FUNCTION_BLOCK print
  (* Standard: 61499-2 *)
  (* Version 0.1, 2018-00-07, hpea485, UOA *)
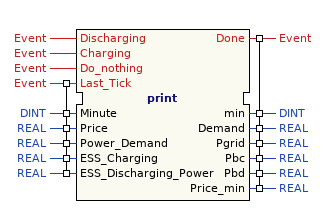
  EVENT_INPUT
    Discharging;
    Charging;
    Do_nothing;
    Last_Tick WITH Minute, Price, Power_Demand, ESS_Charging, ESS_Discharging_Power;
  END_EVENT
  EVENT_OUTPUT
    Done WITH min, Demand, Pgrid, Pbc, Pbd, Price_min;
  END_EVENT
  VAR_INPUT
    Minute : DINT;
    Price : REAL;
    Power_Demand : REAL;
    ESS_Charging : REAL;
    ESS_Discharging_Power : REAL;
  END_VAR
  VAR_OUTPUT
    min : DINT;
    Demand : REAL;
    Pgrid : REAL;
    Pbc : REAL;
    Pbd : REAL;
    Price_min : REAL;
  END_VAR
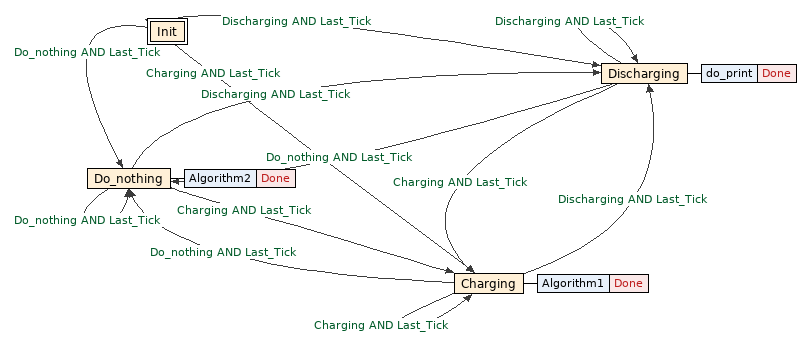
  EC_STATES
    Init;
    Do_nothing : Algorithm2 -> Done;
    Discharging : do_print -> Done;
    Charging : Algorithm1 -> Done;
  END_STATES
  EC_TRANSITIONS
    Do_nothing TO Discharging := Discharging AND Last_Tick;
    Do_nothing TO Charging := Charging AND Last_Tick;
    Do_nothing TO Do_nothing := Do_nothing AND Last_Tick;
    Discharging TO Charging := Charging AND Last_Tick;
    Discharging TO Do_nothing := Do_nothing AND Last_Tick;
    Discharging TO Discharging := Discharging AND Last_Tick;
    Charging TO Discharging := Discharging AND Last_Tick;
    Charging TO Do_nothing := Do_nothing AND Last_Tick;
    Charging TO Charging := Charging AND Last_Tick;
    Init TO Do_nothing := Do_nothing AND Last_Tick;
    Init TO Discharging := Discharging AND Last_Tick;
    Init TO Charging := Charging AND Last_Tick;
  END_TRANSITIONS
  ALGORITHM do_print IN C:
REAL ESS = me->ESS_Discharging_Power;
REAL Pg = me->Power_Demand - ESS;
REAL Power_Demand = me->Power_Demand;
REAL the_price = me->Price;
DINT minute = me->Minute;
printf("Minute in soc do_print %d \r\n", minute);
printf("the price do_print %f \r\n", the_price);
//if (Power_Demand == ESS){
//the_price = 0;
//}
//else if(Power_Demand == Pg){
//the_price = Pg * me->Price;
//}
me->min = minute;
me->Demand = Power_Demand;
me->Pgrid= Pg;
me->Pbc = 0;
me->Pbd = ESS;
me->Price_min = the_price / (30* 2* 1000);// converting $/Mwh to $/kwmin

printf("--------OUTPUT DISCHARGING STATE ------  \r\n");
//printf("DONE \r\n");
printf("Current Minute: %d\tCurrent Price:%f\r\n", me->Minute, the_price);
  END_ALGORITHM
  ALGORITHM Algorithm1 IN C:
REAL the_price = me->Price;
REAL ESS = 200;
REAL Pg = me->Power_Demand + ESS;
REAL Power_Demand = me->Power_Demand;
DINT minute = me->Minute;

me->min = minute;
me->Demand = Power_Demand;
me->Pgrid= Pg;
me->Pbc = ESS;
me->Pbd = 0;
me->Price_min = the_price / (30* 2* 1000);// converting $/Mwh to $/kwmin
printf("Minute in soc al1 %d \r\n", minute);


printf("-------- OUTPUT CHARGING STATE ----- \r\n");
printf("DONE \r\n");

//printf("Current Minute: %d\t Current Price:%f\r\n", me->Minute, me->Price);

//the_price = (Pg + ESS) * me->Price/(2*1000);//price / half kwh *1000
//printf(" Grid POWER: %f \t ESS Power:%f \r\n", Pg, ESS);
printf("Power demand: %f\t Current Price:%f\r\n", me->Power_Demand, the_price);
  END_ALGORITHM
  ALGORITHM Algorithm2 IN C:
REAL the_price = me->Price;
REAL ESS = 200;
REAL Pg = me->Power_Demand + ESS;
REAL Power_Demand = me->Power_Demand;
DINT minute = me->Minute;
printf("Minute in soc al2 %d \r\n", minute);

me->min = minute;
me->Demand = Power_Demand;
me->Pgrid= Power_Demand;
me->Pbc = 0;
me->Pbd = 0;
me->Price_min = the_price / (30* 2* 1000);// converting $/Mwh to $/kwmin

printf("----------NO CHARGE__NO DISCHARGE--------------- \r\n");
printf("DONE \r\n");
printf("Power Demand : %f\t Current Price:%f\r\n", Power_Demand, the_price);
  END_ALGORITHM
END_FUNCTION_BLOCK
